FUNCTION_BLOCK FB_EtherCATFrameDiag
VAR_INPUT
    nFrmXWcState 		: WORD;				// FrmXWcState
    nReqZeroMask 		: WORD := 16#FFFF;	// mask, bit TRUE: require wFrmXWcState.bit = FALSE, bit FALSE: ignore wFrmXWcState.bit *)
END_VAR
VAR_OUTPUT
    bFrameWcStateOK		: BOOL;				// result of fram state check
END_VAR
VAR
END_VAR

(* mask out ignored error bits and compare result against 0 *)
bFrameWcStateOK := ((nFrmXWcState AND nReqZeroMask) = 0);

END_FUNCTION_BLOCK

(* stored: Version 1.1.0.1
   POU FB_EtherCATFrameDiag: Id {c00b03c3-5a7a-47db-a857-8e703b702b2a}, SpecialFunc None *)
